FUNCTION_BLOCK BLOCK_CLIGNOTANT_V0_0
VAR_INPUT
	IN_On:				BOOL;			(*demande de marche*)
END_VAR

VAR_INPUT PERSISTENT
	CONF_Period_On:		TIME:= T#2S;	(*durée de maintien d'allumage*)	
	CONF_Period_Off:	TIME:= T#2S;	(*durée de l'arrêt d'allumage*)
END_VAR

VAR_OUTPUT
	STATE_ON:			BOOL;			(*allumage*)
END_VAR

VAR
	TIMER_On:			TP;
	TIMER_Off:			TP;
END_VAR

TIMER_On.PT		:=	CONF_Period_On;
TIMER_On.IN		:=	IN_On
					AND NOT TIMER_Off.Q;
TIMER_On();

TIMER_Off.PT	:=	CONF_Period_Off;
TIMER_Off.IN	:=	IN_On
					AND NOT TIMER_On.Q;
TIMER_Off();

STATE_ON		:=	TIMER_On.Q and IN_On;

END_FUNCTION_BLOCK

(* stored: Version 1.1.0.1, ProductVersion 3.1.4024.12
   POU BLOCK_CLIGNOTANT_V0_0: Id {e2eeb183-5195-4af4-813e-ad3f9f70bd7f}, SpecialFunc None *)
